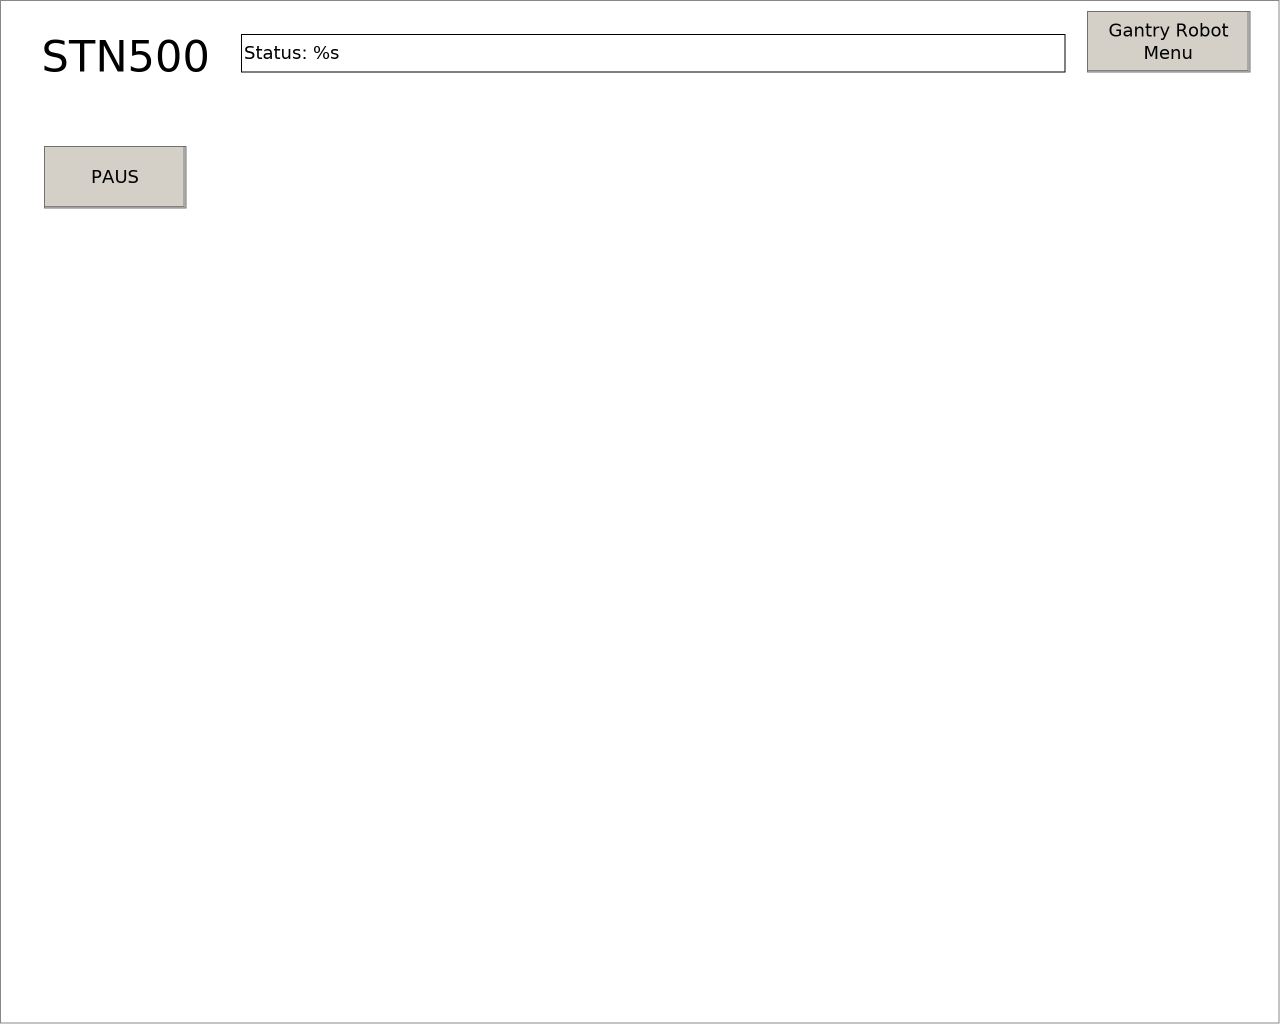
VISUALIZATION Visualization  // 1280x1024
    Label (18,0 216x113), "STN500"
    Button (1087,11 163x61), "Gantry Robot Menu"
        OnMouseClick: change screen: GantryRobotVisu
    Rectangle (241,34 824x38), "Status: %s", text variable: PLC_PRG.fbGantryStatus.Status
    Button (44,146 142x62), "PAUS", input disabled if: NOT PLC_PRG.mxAuto
        toggle PLC_PRG.mxButtonPaus
END_VISUALIZATION

(* stored: Version 1.1.0.1, ProductVersion 3.1.4022.12
   Visu Visualization: Id {866203fd-76f7-4625-b539-f4e49690749e} *)
